FUNCTION_BLOCK FB_Axis
VAR_INPUT
	En: BOOL;
END_VAR

VAR_OUTPUT
	EnO: BOOL;
END_VAR
VAR_IN_OUT
	stAxisStruct						: ST_AxisStruct;
END_VAR
VAR
	fbCommStateMachine			: FB_Communication;
	fbDriveVirtual				: FB_DriveVirtual_V2;
END_VAR

EnO:=En;
fbCommStateMachine(En:=TRUE,
	EnO=> , 
	stAxisStruct:= stAxisStruct);

fbDriveVirtual(En:= TRUE,
	EnO=> ,
	stAxisStruct:=stAxisStruct);

END_FUNCTION_BLOCK

(* stored: Version 1.1.0.1, ProductVersion 3.1.4022.17
   POU FB_Axis: Id {4b9e9ace-3043-48df-9fdf-571ce181897a}, SpecialFunc None *)
